# EPICS StreamDevice protocol: streamDevice/diode.proto
# DolphinDAQ photodiode protocol file
# Built by examining examples at: https://paulscherrerinstitute.github.io/StreamDevice/protocol.html#gen
# And also by examining input/output formats at https://paulscherrerinstitute.github.io/StreamDevice/formats.html

# TODO: Implement the YARR

Terminator = CR LF;

##### Common #####

info {
	ExtraInput = Ignore;
	out "*IDN?";
	in "%39c";
}

debug {
   ExtraInput = Ignore;
   out "%s";
   in "%39c";
}

CountQ {
        out ":TRIGger:COUNt?";
        in "%u";
    }

Count {
        out ":TRIGger:COUNt %u";
        @init { CountQ; }
    }

DecimationQ {
        out ":TRIGger:DECimation?";
        in "%u";
    }

Decimation {
        out ":TRIGger:DECimation %u";
        @init { DecimationQ; }
    }

TimeQ {
        out ":SYSTem:TIME?";
	    in "%39c";
    }

TimeUnixQ {
        out ":SYSTem:TIME:UNIX?";
        in "%i";
    }

TimeUnix {
        out ":SYSTem:TIME:UNIX %i";
        @init { TimeUnixQ; }
    }

##### Diode-Specific #####

TraceDecQ {
        out ":DIODe:TRACe:DECimation?";
        in "%u";
    }

TraceDec {
        out ":DIODe:TRACe:DECimation %u";
        @init { TraceDecQ; }
    }

TraceDtQ {
        out ":DIODe:TRAce:DT?";
        in "%f";
    }

TraceNtQ {
        out ":DIODe:TRAce:NT?";
        in "%f";
    }

TraceYminQ {
        out ":DIODe:TRAce:YMIN?";
        in "%f";
    }

TraceYmaxQ {
        out ":DIODe:TRAce:YMAX?";
        in "%f";
    }

### TODO: TraceYarrayQ {
#        out ":DIODe:TRAce:YARRay?";
#        in "%f";
#    }

DtQ {
        out ":DIODe:DT?";
        in "%f";
    }

Dt {
        out ":DIODE:DT %i";
    }

T1NtQ {
        out ":DIODE:T3:NT?";
        in "%u";
    }

T1Q {
        out ":DIODE:T1:VALue?";
        in "%f";
    }

T1 {
        out ":DIODE:T1:VALue %f";
        @init { T1Q; }
    }

T2NtQ {
        out ":DIODE:T2:NT?";
        in "%u";
    }

T2Q {
        out ":DIODE:T2:VALue?";
        in "%f";
    }

T2 {
        out ":DIODE:T2:VALue %f";
        @init { T2Q; }
    }

T3NtQ {
        out ":DIODE:T3:NT?";
        in "%u";
    }

T3Q {
        out ":DIODE:T3:VALue?";
        in "%f";
    }

T3 {
        out ":DIODE:T3:VALue %f";
        @init { T3Q; }
    }

T4NtQ {
        out ":DIODE:T4:NT?";
        in "%u";
    }

T4Q {
        out ":DIODE:T4:VALue?";
        in "%f";
    }

T4 {
        out ":DIODE:T4:VALue %f";
        @init { T4Q; }
    }
